INTERFACE I_Machine

METHOD Config : BOOL
VAR_INPUT
	stConfig: ST_Config;
END_VAR
END_METHOD

METHOD MoveNext : BOOL
VAR_INPUT
END_VAR
END_METHOD

METHOD Start : BOOL
VAR_INPUT
END_VAR
END_METHOD

END_INTERFACE

(* stored: Version 1.1.0.1, ProductVersion 3.1.4024.3
   Itf I_Machine: Id {7529e6e0-a30a-4fae-ad5c-493ba6237ce4}
   Method Config: Id {297ce5e8-35f5-447a-9541-fe4a8ddfe9de}
   Method MoveNext: Id {c78f4b92-86b9-4159-8d15-ffc912641fd0}
   Method Start: Id {71cb3e41-c453-4a91-8dbb-66ee27c55389} *)
